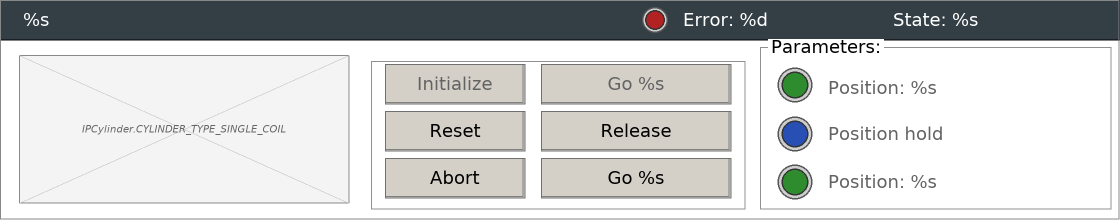
VISUALIZATION SingleCylinder  // 1120x220
VAR_IN_OUT
	stCylinder : ST_VisuCtrlCylinderFrame;
END_VAR
    Rectangle (0,0 1120x40)
    Textfield (20,5 524x30), "%s", text variable: stCylinder.sName
    Textfield (890,5 225x30), "State: %s", text list: 'TL_SingleCylinderState', text index: stCylinder.eCylinderState
    Lamp1 (640,5 30x30), variable: stCylinder.bError, style: Lamp-Lamp1-Red
    Textfield (680,5 200x30), "Error: %d", text variable: stCylinder.iErrorID
    GroupBox (760,39 351x170), "Parameters:"
        Rectangle (65,85 270x20), "Position hold", text variable: stCylinder.sHomeDescription
        Lamp1 (15,75 40x40), variable: stCylinder.bPositionHold, style: Lamp-Lamp1-Blue
        Rectangle (65,133 270x20), "Position: %s", text variable: stCylinder.sHomeDescription
        Rectangle (65,39 270x20), "Position: %s", text variable: stCylinder.sActiveDescription
        Lamp1 (15,26 40x40), variable: stCylinder.bSensorActive, style: Lamp-Lamp1-Green
        Lamp1 (15,123 40x40), variable: stCylinder.bSensorHome, style: Lamp-Lamp1-Green
    GroupBox (371,53 374x156)
        Button (170,105 190x40), "Go %s", text variable: stCylinder.sHomeDescription
            tap stCylinder.btnGoHome
        Button (170,58 190x40), "Release"
            tap stCylinder.btnRealase
        Button (170,11 190x40), "Go %s", text variable: stCylinder.sActiveDescription
            tap stCylinder.btnGoActive
        Button (14,105 140x40), "Abort", text variable: stCylinder.sHomeDescription
            tap stCylinder.btnAbort
        Button (14,58 140x40), "Reset"
            tap stCylinder.btnReset
        Button (14,11 140x40), "Initialize", text variable: stCylinder.sActiveDescription
            tap stCylinder.btnInit
    Image (19,55 330x148), image: IPCylinder.CYLINDER_TYPE_SINGLE_COIL
        p84334746: stCylinder.sCylinderImage
END_VISUALIZATION

(* stored: Version 1.1.0.1, ProductVersion 3.1.4024.9
   Visu SingleCylinder: Id {8e55db11-d66c-4ad5-88f4-1c04ab6235e6} *)
